// TIA Portal V20 export
VAR_GLOBAL   // PLC tag table "Unit1Em0"
   "BA060ZSIBK04.00" AT %I1012.0 : Bool;   // (HOME) STACK #1 NG CLAMP MOVER OPEN
   "BA060ZSIBK04.02" AT %I1012.2 : Bool;   // (HOME) STACK #1 NG CLAMP LEFT OPEN
   "BA060ZSIBK04.01" AT %I1012.1 : Bool;   // (HOME) STACK #1 NG CLAMP RIGHT OPEN
   "BA060ZSIBK04.03" AT %I1012.3 : Bool;   // (HOME) STAKC #1 NG CLAMP Z-AXIS UP
   "BA060ZSIBK04.04" AT %I1012.4 : Bool;   // (HOME) STAKC #1 NG CLAMP MOVER BACKWARD
   "BA060ZSIBK04.05" AT %I1012.5 : Bool;   // (HOME) STACK #1 NG BOX LIFT DOWN
   "BA060ZSIBK04.06" AT %I1012.6 : Bool;   // (HOME) STACK #1 NG BOX LOCK DOWN
   "BA060ZSIBK04.07" AT %I1012.7 : Bool;   // STACK 1 NG BOX FULL SENSOR
   "BA060ZSIBK04.08" AT %I1013.0 : Bool;   // (WORK) STACK #1 NG CLAMP MOVER CLOSE
   "BA060ZSIBK04.10" AT %I1013.2 : Bool;   // (WORK) STACK #1 NG CLAMP LEFT CLOSE
   "BA060ZSIBK04.09" AT %I1013.1 : Bool;   // (WORK) STACK #1 NG CLAMP RIGHT CLOSE
   "BA060ZSIBK04.11" AT %I1013.3 : Bool;   // (WORK) STAKC #1 NG CLAMP Z-AXIS DOWN
   "BA060ZSIBK04.12" AT %I1013.4 : Bool;   // (WORK) STAKC #1 NG CLAMP MOVER FORWARD
   "BA060ZSIBK04.13" AT %I1013.5 : Bool;   // (WORK) STACK #1 NG BOX LIFT UP
   "BA060ZSIBK04.14" AT %I1013.6 : Bool;   // (WORK) STACK #1 NG BOX LOCK UP
   "BA060ZSIBK04.15" AT %I1013.7 : Bool;   // SPARE
   "BA060ZSIBK01.04" AT %I1000.4 : Bool;   // STACK 1 NG BOX DETECT SENSOR
   "BA060ZSIPM01.00" AT %Q2000.0 : Bool;   // (WORK) STACK #1 NG CLAMP MOVER CLOSE
   "BA060ZSIPM01.01" AT %Q2000.1 : Bool;   // (HOME) STACK #1 NG CLAMP MOVER OPEN
   "BA060ZSIPM01.02" AT %Q2000.2 : Bool;   // (WORK) STACK #1 NG CLAMP RIGHT CLOSE
   "BA060ZSIPM01.03" AT %Q2000.3 : Bool;   // (HOME) STACK #1 NG CLAMP RIGHT OPEN
   "BA060ZSIPM01.04" AT %Q2000.4 : Bool;   // (HOME) STACK #1 NG CLAMP LEFT OPEN
   "BA060ZSIPM01.05" AT %Q2000.5 : Bool;   // (WORK) STACK #1 NG CLAMP LEFT CLOSE
   "BA060ZSIPM01.06" AT %Q2000.6 : Bool;   // (HOME) STAKC #1 NG CLAMP Z-AXIS UP
   "BA060ZSIPM01.07" AT %Q2000.7 : Bool;   // (WORK) STAKC #1 NG CLAMP Z-AXIS DOWN
   "BA060ZSIPM01.10" AT %Q2001.0 : Bool;   // (WORK) STAKC #1 NG CLAMP MOVER FORWARD
   "BA060ZSIPM01.11" AT %Q2001.1 : Bool;   // (HOME) STAKC #1 NG CLAMP MOVER BACKWARD
   "BA060ZSIPM01.12" AT %Q2001.2 : Bool;   // (WORK) STACK #1 NG BOX LIFT UP
   "BA060ZSIPM01.13" AT %Q2001.3 : Bool;   // (HOME) STACK #1 NG BOX LIFT DOWN
   "BA060ZSIPM01.14" AT %Q2001.4 : Bool;   // (WORK) STACK #1 NG BOX LOCK UP
   "BA060ZSIPM01.15" AT %Q2001.5 : Bool;   // (HOME) STACK #1 NG BOX LOCK DOWN
END_VAR
VAR_GLOBAL CONSTANT   // user constants
   U1EM0_JOB01 : DInt := 1;
   U1EM0_JOB02 : DInt := 2;
   U1EM0_JOB03 : DInt := 3;
   U1EM0_JOB04 : DInt := 4;
   U1EM0_JOB05 : DInt := 5;
   U1EM0_JOB06 : DInt := 6;
   U1EM0_JOB07 : DInt := 7;
   U1EM0_JOB08 : DInt := 8;
   U1EM0_JOB09 : DInt := 9;
   U1EM0_JOB10 : DInt := 10;
   U1EM0_JOB11 : DInt := 11;
   U1EM0_JOB12 : DInt := 12;
   U1EM0_JOB13 : DInt := 13;
   U1EM0_JOB14 : DInt := 14;
   U1EM0_JOB15 : DInt := 15;
   U1EM0_JOB16 : DInt := 16;
   U1EM0_JOB17 : DInt := 17;
   U1EM0_JOB18 : DInt := 18;
   U1EM0_JOB19 : DInt := 19;
   U1EM0_JOB20 : DInt := 20;
   U1EM0_JOB21 : DInt := 21;
   U1EM0_JOB22 : DInt := 22;
   U1EM0_JOB23 : DInt := 23;
   U1EM0_JOB24 : DInt := 24;
   U1EM0_JOB25 : DInt := 25;
   U1EM0_JOB26 : DInt := 26;
   U1EM0_JOB27 : DInt := 27;
   U1EM0_JOB28 : DInt := 28;
   U1EM0_JOB29 : DInt := 29;
   U1EM0_JOB30 : DInt := 30;
   U1EM0_JOB31 : DInt := 31;
   U1EM0_JOB32 : DInt := 32;
   U1EM0_JOB33 : DInt := 33;
   U1EM0_JOB34 : DInt := 34;
   U1EM0_JOB35 : DInt := 35;
   U1EM0_JOB36 : DInt := 36;
   U1EM0_JOB37 : DInt := 37;
   U1EM0_JOB38 : DInt := 38;
   U1EM0_JOB39 : DInt := 39;
   U1EM0_JOB40 : DInt := 40;
   U1EM0_JOB41 : DInt := 41;
   U1EM0_JOB42 : DInt := 42;
   U1EM0_JOB43 : DInt := 43;
   U1EM0_JOB44 : DInt := 44;
   U1EM0_JOB45 : DInt := 45;
   U1EM0_JOB46 : DInt := 46;
   U1EM0_JOB47 : DInt := 47;
   U1EM0_JOB48 : DInt := 48;
   U1EM0_JOB49 : DInt := 49;
   U1EM0_JOB50 : DInt := 50;
   U1EM0_JOB51 : DInt := 51;
   U1EM0_JOB52 : DInt := 52;
   U1EM0_JOB53 : DInt := 53;
   U1EM0_JOB54 : DInt := 54;
   U1EM0_JOB55 : DInt := 55;
   U1EM0_JOB56 : DInt := 56;
   U1EM0_JOB57 : DInt := 57;
   U1EM0_JOB58 : DInt := 58;
   U1EM0_JOB59 : DInt := 59;
   U1EM0_JOB60 : DInt := 60;
   U1EM0_JOB61 : DInt := 61;
   U1EM0_JOB62 : DInt := 62;
   U1EM0_JOB63 : DInt := 63;
   U1EM0_JOB64 : DInt := 64;
   U1EM0_JOB65 : DInt := 65;
   U1EM0_JOB66 : DInt := 66;
   U1EM0_JOB67 : DInt := 67;
   U1EM0_JOB68 : DInt := 68;
   U1EM0_JOB69 : DInt := 69;
   U1EM0_JOB70 : DInt := 70;
   U1EM0_JOB71 : DInt := 71;
   U1EM0_JOB72 : DInt := 72;
   U1EM0_JOB73 : DInt := 73;
   U1EM0_JOB74 : DInt := 74;
   U1EM0_JOB75 : DInt := 75;
   U1EM0_JOB76 : DInt := 76;
   U1EM0_JOB77 : DInt := 77;
   U1EM0_JOB78 : DInt := 78;
   U1EM0_JOB79 : DInt := 79;
   U1EM0_JOB80 : DInt := 80;
   U1EM0_JOB81 : DInt := 81;
   U1EM0_JOB82 : DInt := 82;
   U1EM0_JOB83 : DInt := 83;
   U1EM0_JOB84 : DInt := 84;
   U1EM0_JOB85 : DInt := 85;
   U1EM0_JOB86 : DInt := 86;
   U1EM0_JOB87 : DInt := 87;
   U1EM0_JOB88 : DInt := 88;
   U1EM0_JOB89 : DInt := 89;
   U1EM0_JOB90 : DInt := 90;
   U1EM0_JOB91 : DInt := 91;
   U1EM0_JOB92 : DInt := 92;
   U1EM0_JOB93 : DInt := 93;
   U1EM0_JOB94 : DInt := 94;
   U1EM0_JOB95 : DInt := 95;
   U1EM0_JOB96 : DInt := 96;
   U1EM0_JOB97 : DInt := 97;
   U1EM0_JOB98 : DInt := 98;
   U1EM0_JOB99 : DInt := 99;
   U1EM0_SEQUENCE01 : Int := 1;
   U1EM0_SEQUENCE02 : Int := 2;
   U1EM0_SEQUENCE03 : Int := 3;
   U1EM0_SEQUENCE04 : Int := 4;
   U1EM0_SEQUENCE05 : Int := 5;
   U1EM0_SEQUENCE06 : Int := 6;
   U1EM0_SEQUENCE07 : Int := 7;
   U1EM0_SEQUENCE08 : Int := 8;
   U1EM0_SEQUENCE09 : Int := 9;
   U1EM0_SEQUENCE10 : Int := 10;
   U1EM0_SEQUENCE11 : Int := 11;
   U1EM0_SEQUENCE12 : Int := 12;
   U1EM0_SEQUENCE13 : Int := 13;
   U1EM0_SEQUENCE14 : Int := 14;
   U1EM0_SEQUENCE15 : Int := 15;
   U1EM0_SEQUENCE16 : Int := 16;
   U1EM0_SEQUENCE17 : Int := 17;
   U1EM0_SEQUENCE18 : Int := 18;
   U1EM0_SEQUENCE19 : Int := 19;
   U1EM0_SEQUENCE20 : Int := 20;
   U1EM0_SEQUENCE21 : Int := 21;
   U1EM0_SEQUENCE22 : Int := 22;
   U1EM0_SEQUENCE23 : Int := 23;
   U1EM0_SEQUENCE24 : Int := 24;
   U1EM0_SEQUENCE25 : Int := 25;
   U1EM0_SEQUENCE26 : Int := 26;
   U1EM0_SEQUENCE27 : Int := 27;
   U1EM0_SEQUENCE28 : Int := 28;
   U1EM0_SEQUENCE29 : Int := 29;
   U1EM0_SEQUENCE30 : Int := 30;
   U1EM0_SEQUENCE31 : Int := 31;
   U1EM0_SEQUENCE32 : Int := 32;
   U1EM0_SEQUENCE33 : Int := 33;
   U1EM0_SEQUENCE34 : Int := 34;
   U1EM0_SEQUENCE35 : Int := 35;
   U1EM0_SEQUENCE36 : Int := 36;
   U1EM0_SEQUENCE37 : Int := 37;
   U1EM0_SEQUENCE38 : Int := 38;
   U1EM0_SEQUENCE39 : Int := 39;
   U1EM0_SEQUENCE40 : Int := 40;
   U1EM0_SEQUENCE41 : Int := 41;
   U1EM0_SEQUENCE42 : Int := 42;
   U1EM0_SEQUENCE43 : Int := 43;
   U1EM0_SEQUENCE44 : Int := 44;
   U1EM0_SEQUENCE45 : Int := 45;
   U1EM0_SEQUENCE46 : Int := 46;
   U1EM0_SEQUENCE47 : Int := 47;
   U1EM0_SEQUENCE48 : Int := 48;
   U1EM0_SEQUENCE49 : Int := 49;
   U1EM0_SEQUENCE50 : Int := 50;
   U1EM0_SEQUENCE51 : Int := 51;
   U1EM0_SEQUENCE52 : Int := 52;
   U1EM0_SEQUENCE53 : Int := 53;
   U1EM0_SEQUENCE54 : Int := 54;
   U1EM0_SEQUENCE55 : Int := 55;
   U1EM0_SEQUENCE56 : Int := 56;
   U1EM0_SEQUENCE57 : Int := 57;
   U1EM0_SEQUENCE58 : Int := 58;
   U1EM0_SEQUENCE59 : Int := 59;
   U1EM0_SEQUENCE60 : Int := 60;
   U1EM0_SEQUENCE61 : Int := 61;
   U1EM0_SEQUENCE62 : Int := 62;
   U1EM0_SEQUENCE63 : Int := 63;
   U1EM0_SEQUENCE64 : Int := 64;
   U1EM0_SEQUENCE65 : Int := 65;
   U1EM0_SEQUENCE66 : Int := 66;
   U1EM0_SEQUENCE67 : Int := 67;
   U1EM0_SEQUENCE68 : Int := 68;
   U1EM0_SEQUENCE69 : Int := 69;
   U1EM0_SEQUENCE70 : Int := 70;
   U1EM0_SEQUENCE71 : Int := 71;
   U1EM0_SEQUENCE72 : Int := 72;
   U1EM0_SEQUENCE73 : Int := 73;
   U1EM0_SEQUENCE74 : Int := 74;
   U1EM0_SEQUENCE75 : Int := 75;
   U1EM0_SEQUENCE76 : Int := 76;
   U1EM0_SEQUENCE77 : Int := 77;
   U1EM0_SEQUENCE78 : Int := 78;
   U1EM0_SEQUENCE79 : Int := 79;
   U1EM0_SEQUENCE80 : Int := 80;
   U1EM0_SEQUENCE81 : Int := 81;
   U1EM0_SEQUENCE82 : Int := 82;
   U1EM0_SEQUENCE83 : Int := 83;
   U1EM0_SEQUENCE84 : Int := 84;
   U1EM0_SEQUENCE85 : Int := 85;
   U1EM0_SEQUENCE86 : Int := 86;
   U1EM0_SEQUENCE87 : Int := 87;
   U1EM0_SEQUENCE88 : Int := 88;
   U1EM0_SEQUENCE89 : Int := 89;
   U1EM0_SEQUENCE90 : Int := 90;
   U1EM0_SEQUENCE91 : Int := 91;
   U1EM0_SEQUENCE92 : Int := 92;
   U1EM0_SEQUENCE93 : Int := 93;
   U1EM0_SEQUENCE94 : Int := 94;
   U1EM0_SEQUENCE95 : Int := 95;
   U1EM0_SEQUENCE96 : Int := 96;
   U1EM0_SEQUENCE97 : Int := 97;
   U1EM0_SEQUENCE98 : Int := 98;
   U1EM0_SEQUENCE99 : Int := 99;
   U1EM0_NO_OF_SEQUENCE : Int := 1;
END_VAR
